// TIA Portal V16 export
// export: Created 2023-03-29T11:03:22.6082356Z, ExportSetting WithDefaults, DisplayName Totally Integrated Automation Portal, DisplayVersion V16 Update 6, DisplayName TIA Portal Version Control Interface, DisplayVersion V16 Update 2, DisplayName TIA Portal Openness, DisplayVersion V16 Update 6, DisplayName STEP 7 Professional, DisplayVersion V16 Update 6, DisplayName STEP 7 Safety, DisplayVersion V16, DisplayName WinCC Advanced, DisplayVersion V16 Update 6
FUNCTION "Sterowanie_Zbiornik" : Void   // FC26, LAD
TITLE = Napełnianie i opróżnianie
{ S7_Optimized_Access := 'TRUE' }
AUTHOR : rtecmer
VERSION : 0.1
// Funkcja steruje napędami napełniania i opróżniania w cyklu od zegara czasu jak i od pomiaru poziomu. Poziom jest sygnałem nadrzędnym. Jeśli napełnienie uzyskano przed czasem to napełnianie jest kończone z osiągnięciem poziomu max. Podczas oróżniania jeśli osiągnięto poziom min to opróżnianie zbiorniak jest zakończone.
// Granica końca minimum to 100cm ponad tę wartość nastąpi dopiero skasowanie sygnału poziom MIN
// Spadku poziomu poniżej 250cm pozwala na scasowanie sygnału poziom MAX
// stored: AutoNumber true, IsIECCheckEnabled false, SetENOAutomatically false, UDAEnableTagReadback false
   VAR_INPUT
      actLevel : Real;   // pozim w zbiorniku
      maxLevel : Real;   // poziom napełnienia
      minLevel : Real;   // poziom opróżnienia
      actTime : Real;   // czas aktualny
      actTime_FillingOn : Real;   // godzina start napełnianie
      actTime_FillingOff : Real;   // godzina stop napełnianie
      actTime_EmptyingOn : Real;   // godzina start przetłaczanie
      actTime_EmptyingOff : Real;   // godzina stop przetłaczanie
      isOpen_filling : Bool;   // potwierdzenie otwarcia napełniającej zasuwy
      isOpen_emptying : Bool;   // potwierdzenie otwarcia spustowej zasuwy
      isClose_filling : Bool;   // potwierdzenie zamknięcia napełniającej zasuwy
      isClose_emptying : Bool;   // potwierdzenie zamknięcia spustowej zasuwy
      isReady_filling : Bool;   // sygnał gotowości zasuwa napełnianie
      isReadyt_emptying : Bool;   // sygnał gotowości zasuwa spustowa
      activTank : Bool;   // zbiornik aktywny
      isAut_Valve_Filling : Bool;   // tryb pracy automat zasuwa napełnianie
      isAut_Valve_Empting : Bool;   // tryb pracy automat zasuwa spustowa
      is_min_Float : Bool;   // sygnał minimum z płyawaka
      is_max_Float : Bool;   // sygnał max z płyawaka
      isAlarmNinimum_barB5 : Bool;   // alarm niskie ciśnienie magistrala
      resetAlarmMinimum_barB5 : Bool;   // koniec alarm niskie ciśnienie magistral
      setTank_Work_daily : Bool;   // tryb pracy dobowy aktywny
      setTank_Work_selective : Bool;   // tryb pracy selektywny - jeden zbiornik aktywny
      setControl_alarm_B5 : Bool;   // sygnał uruchomienie awaryjnego otwarcie zbiornika na dosilanie
      set_HWork_tank : Bool;   // ustawia aktywny zbiornik do pracy w trybie selektywnym
   END_VAR
   VAR_OUTPUT
      setSVMO_Z_Wlot : Bool;   // bit otwierania w trybie automat
      setSVMC_Z_Wlot : Bool;   // bit zamykania w trybie automat
      setSVMO_Z_Spust : Bool;   // bit otwierania w trybie automat
      setSVMC_Z_Spust : Bool;   // bit zamykania w trybie automat
      infoFiling_to_HMI : Bool;   // bit informacji wejściu w tryb napełniania
   END_VAR
   VAR_IN_OUT
      isFilling : Bool;   // bit aktywacji napełninia
      isEptying : Bool;   // bit aktywacji przetłaczania
      memRisingLevel_min : Bool;   // pamięc zbocza osiągniecia poziomu minimum w zbiorniku
      memRisingLevel_max : Bool;   // pamięc zbocza osiągniecia poziomu max w zbiorniku
      isLevelMax : Bool;   // poziom max
      isLevelMin : Bool;   // poziom min
      blok_tank : Bool;   // bit blokowania zbiornika w sekwencji
   END_VAR
   VAR_TEMP
      correction_max : Real;   // współczynnik korekty dla zachowania histerezy przy wahaniu poziomu w zbiorniku
      correction_min : Real;   // współczynnik korekty dla zachowania histerezy przy wahaniu poziomu w zbiorniku
      filling_time : Real;   // wyliczony czas napełniania na dobę
      filing_time_X : Bool;   // bit logika gdy napełnianie przed 00:00
      filing_time_Y : Bool;   // bit logika gdy napełnianie po 00:01
      epting_time_X : Bool;   // bit logika gdy napełnianie po 00:01
   END_VAR
   VAR_TEMP   // added for the SCL form of the ladder/FBD networks
      _w1 : Bool;
      _w2 : Bool;
   END_VAR
BEGIN

REGION Network 1 (SCL): wyliczenie korekty dla stabilności sygału min i max
   #correction_max := (#maxLevel - 30);
   #correction_min := (#minLevel + 20);
END_REGION

REGION Network 2: znacznik poziom max
   // przechwycenie poziomu max
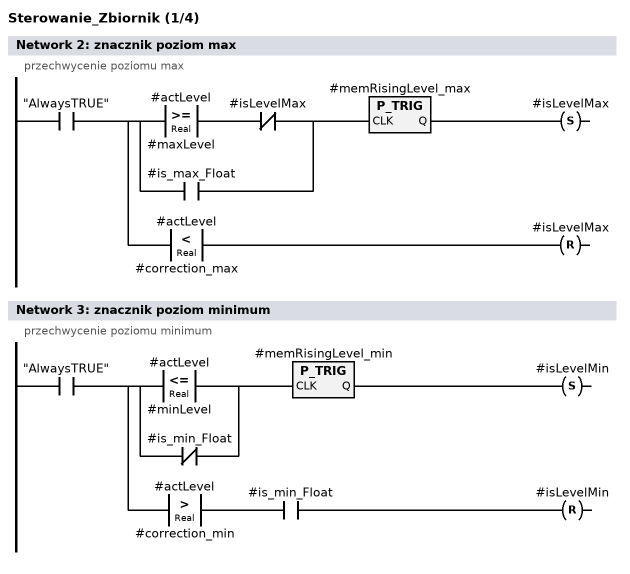
   RUNG wire#powerrail
      Contact( "AlwaysTRUE" )
      wire#w1
      { S7_Templates := "SrcType := Real" } GE_Contact(in1 := #actLevel, in2 := #maxLevel)
      I_Contact( #isLevelMax )
      wire#w2
      P_Trig( #memRisingLevel_max )
      S_Coil( #isLevelMax )
   END_RUNG
   RUNG wire#w1
      Contact( #is_max_Float )
   END_RUNG wire#w2
   RUNG wire#w1
      { S7_Templates := "SrcType := Real" } LT_Contact(in1 := #actLevel, in2 := #correction_max)
      R_Coil( #isLevelMax )
   END_RUNG
   // the same network as SCL:
   #_w1 := "AlwaysTRUE" AND (((#actLevel >= #maxLevel) AND NOT #isLevelMax) OR #is_max_Float);
   #_w2 := #_w1 AND NOT #memRisingLevel_max;   // rising edge
   #memRisingLevel_max := #_w1;
   IF #_w2 THEN #isLevelMax := TRUE; END_IF;
   IF "AlwaysTRUE" AND (#actLevel < #correction_max) THEN #isLevelMax := FALSE; END_IF;
END_REGION

REGION Network 3: znacznik poziom minimum
   // przechwycenie poziomu minimum
   RUNG wire#powerrail
      Contact( "AlwaysTRUE" )
      wire#w1
      { S7_Templates := "SrcType := Real" } LE_Contact(in1 := #actLevel, in2 := #minLevel)
      wire#w2
      P_Trig( #memRisingLevel_min )
      S_Coil( #isLevelMin )
   END_RUNG
   RUNG wire#w1
      I_Contact( #is_min_Float )
   END_RUNG wire#w2
   RUNG wire#w1
      { S7_Templates := "SrcType := Real" } GT_Contact(in1 := #actLevel, in2 := #correction_min)
      Contact( #is_min_Float )
      R_Coil( #isLevelMin )
   END_RUNG
   // the same network as SCL:
   #_w1 := "AlwaysTRUE" AND ((#actLevel <= #minLevel) OR NOT #is_min_Float);
   #_w2 := #_w1 AND NOT #memRisingLevel_min;   // rising edge
   #memRisingLevel_min := #_w1;
   IF #_w2 THEN #isLevelMin := TRUE; END_IF;
   IF "AlwaysTRUE" AND (#actLevel > #correction_min) AND #is_min_Float THEN #isLevelMin := FALSE; END_IF;
END_REGION

REGION Network 4 (SCL): wyliczony czas napełniania na dobę i ustawoanie bitu kontroli pracy w dobie
   // #filing_time_X  - bit ustawiany w przypadku gdy w przedziale pracy wystąpi przejście przez  godzinę 00:00
   IF #actTime_FillingOn > #actTime_FillingOff THEN
     // odejmnij od wiekszej mniejszą
     #filling_time := (#actTime_FillingOn - #actTime_FillingOff);
     IF #actTime >=  #actTime_FillingOn THEN
       // jeśli czas rozpoczęcia napełniania to ustaw bit
       #filing_time_X := TRUE;
       ;
     ELSE
       // w innym wypadku kasuj bit
       #filing_time_X := False;
       ;
     END_IF;

     #filing_time_Y := FALSE;
   ELSE
     #filling_time := (#actTime_FillingOff - #actTime_FillingOn);
     #filing_time_X := False;
     #filing_time_Y := TRUE;
     ;
   END_IF;
END_REGION

REGION Network 5: bit aktywacji napełninia
   // aktywacja, deaktywacja bitu rocedury napełniania
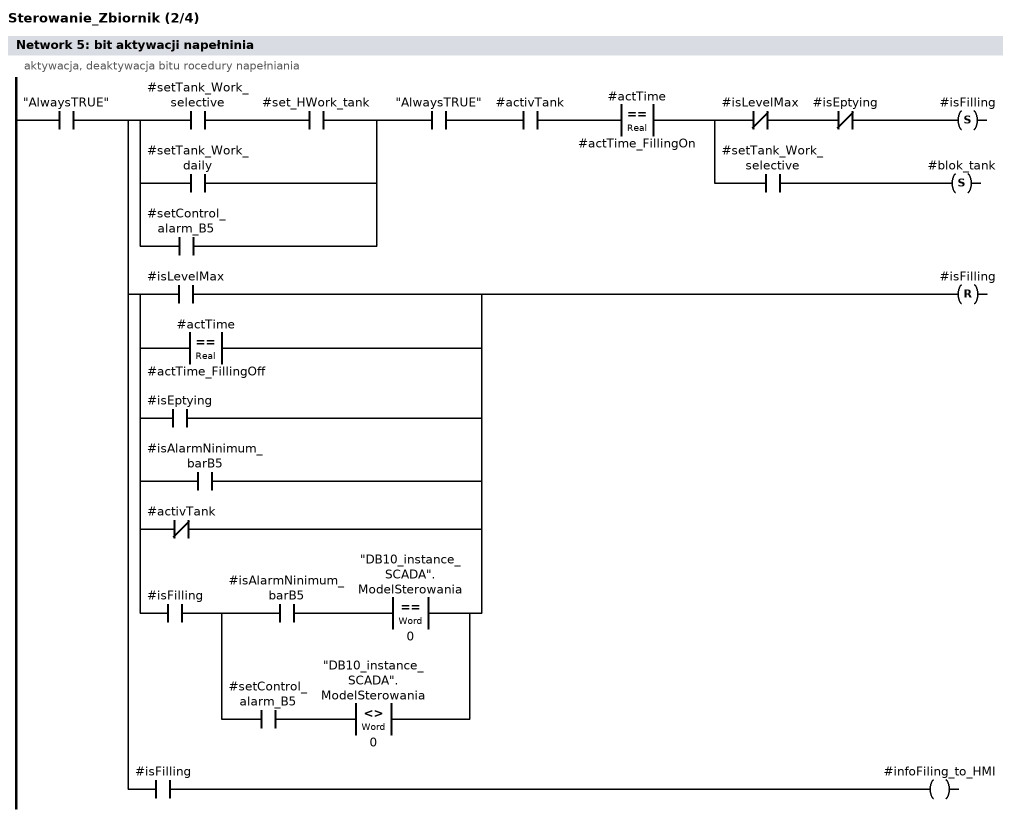
   RUNG wire#powerrail
      Contact( "AlwaysTRUE" )
      wire#w1
      Contact( #setTank_Work_selective )
      Contact( #set_HWork_tank )
      wire#w2
      Contact( "AlwaysTRUE" )
      Contact( #activTank )
      { S7_Templates := "SrcType := Real" } EQ_Contact(in1 := #actTime, in2 := #actTime_FillingOn)
      wire#w3
      I_Contact( #isLevelMax )
      I_Contact( #isEptying )
      S_Coil( #isFilling )
   END_RUNG
   RUNG wire#w1
      Contact( #setTank_Work_daily )
   END_RUNG wire#w2
   RUNG wire#w1
      Contact( #setControl_alarm_B5 )
   END_RUNG wire#w2
   RUNG wire#w3
      Contact( #setTank_Work_selective )
      S_Coil( #blok_tank )
   END_RUNG
   RUNG wire#w1
      Contact( #isLevelMax )
      wire#w4
      R_Coil( #isFilling )
   END_RUNG
   RUNG wire#w1
      { S7_Templates := "SrcType := Real" } EQ_Contact(in1 := #actTime, in2 := #actTime_FillingOff)
   END_RUNG wire#w4
   RUNG wire#w1
      Contact( #isEptying )
   END_RUNG wire#w4
   RUNG wire#w1
      Contact( #isAlarmNinimum_barB5 )
   END_RUNG wire#w4
   RUNG wire#w1
      I_Contact( #activTank )
   END_RUNG wire#w4
   RUNG wire#w1
      Contact( #isFilling )
      wire#w5
      Contact( #isAlarmNinimum_barB5 )
      { S7_Templates := "SrcType := Word" } EQ_Contact(in1 := "DB10_instance_SCADA".ModelSterowania, in2 := 0)
   END_RUNG wire#w4
   RUNG wire#w5
      Contact( #setControl_alarm_B5 )
      { S7_Templates := "SrcType := Word" } NE_Contact(in1 := "DB10_instance_SCADA".ModelSterowania, in2 := 0)
   END_RUNG wire#w4
   RUNG wire#w1
      Contact( #isFilling )
      Coil( #infoFiling_to_HMI )
   END_RUNG
   // the same network as SCL:
   #_w1 := "AlwaysTRUE" AND ((#setTank_Work_selective AND #set_HWork_tank) OR #setTank_Work_daily OR #setControl_alarm_B5) AND "AlwaysTRUE" AND #activTank AND (#actTime = #actTime_FillingOn);
   IF #_w1 AND NOT #isLevelMax AND NOT #isEptying THEN #isFilling := TRUE; END_IF;
   IF #_w1 AND #setTank_Work_selective THEN #blok_tank := TRUE; END_IF;
   IF "AlwaysTRUE" AND (#isLevelMax OR (#actTime = #actTime_FillingOff) OR #isEptying OR #isAlarmNinimum_barB5 OR NOT #activTank OR (#isFilling AND ((#isAlarmNinimum_barB5 AND ("DB10_instance_SCADA".ModelSterowania = 0)) OR (#setControl_alarm_B5 AND ("DB10_instance_SCADA".ModelSterowania <> 0))))) THEN
       #isFilling := FALSE;
   END_IF;
   #infoFiling_to_HMI := "AlwaysTRUE" AND #isFilling;
END_REGION

REGION Network 6 (SCL): ustawoanie bitu kontroli pracy w dobie
   // epting_time_X  - bit ustawiany w przypadku gdy w przedziale pracy wystąpi przejście przez  godzinę 00:00
   IF #actTime_EmptyingOn > #actTime_EmptyingOff THEN

     IF #actTime >=  #actTime_EmptyingOn THEN
       // jeśli czas rozpoczęcia napełniania to ustaw bit
       #epting_time_X := TRUE;
       ;
     ELSE
       // w innym wypadku kasuj bit
       #epting_time_X := False;
       ;
     END_IF;

   ELSE

     #epting_time_X := False;

     ;
   END_IF;
END_REGION

REGION Network 7: bit aktywacji przetłaczania
   // aktywacja/ deaktywacja bitu pracy pompowni (przetłaczanie)
   // musi zakonczyć się napełnianie, jeśli wyłaczysz z trybu automat to reset znacznika przetłaczanie
   // 
   // #epting_time_X - usunąłem na testy
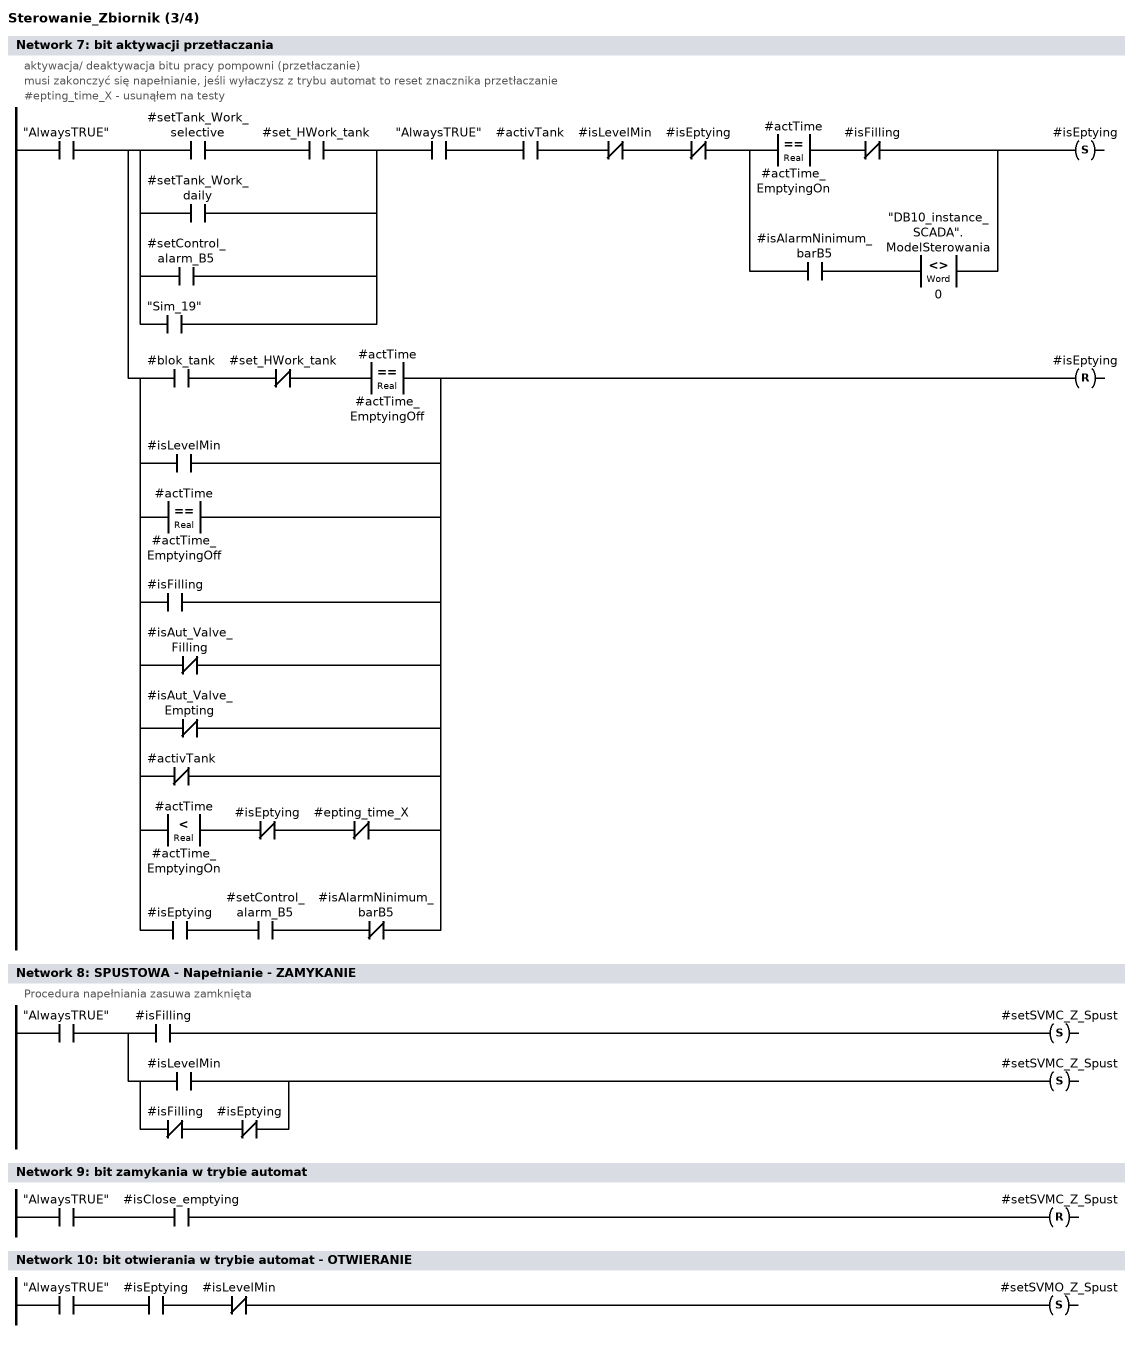
   RUNG wire#powerrail
      Contact( "AlwaysTRUE" )
      wire#w1
      Contact( #setTank_Work_selective )
      Contact( #set_HWork_tank )
      wire#w2
      Contact( "AlwaysTRUE" )
      Contact( #activTank )
      I_Contact( #isLevelMin )
      I_Contact( #isEptying )
      wire#w3
      { S7_Templates := "SrcType := Real" } EQ_Contact(in1 := #actTime, in2 := #actTime_EmptyingOn)
      I_Contact( #isFilling )
      wire#w4
      S_Coil( #isEptying )
   END_RUNG
   RUNG wire#w1
      Contact( #setTank_Work_daily )
   END_RUNG wire#w2
   RUNG wire#w1
      Contact( #setControl_alarm_B5 )
   END_RUNG wire#w2
   RUNG wire#w1
      Contact( "Sim_19" )
   END_RUNG wire#w2
   RUNG wire#w3
      Contact( #isAlarmNinimum_barB5 )
      { S7_Templates := "SrcType := Word" } NE_Contact(in1 := "DB10_instance_SCADA".ModelSterowania, in2 := 0)
   END_RUNG wire#w4
   RUNG wire#w1
      Contact( #blok_tank )
      I_Contact( #set_HWork_tank )
      { S7_Templates := "SrcType := Real" } EQ_Contact(in1 := #actTime, in2 := #actTime_EmptyingOff)
      wire#w5
      R_Coil( #isEptying )
   END_RUNG
   RUNG wire#w1
      Contact( #isLevelMin )
   END_RUNG wire#w5
   RUNG wire#w1
      { S7_Templates := "SrcType := Real" } EQ_Contact(in1 := #actTime, in2 := #actTime_EmptyingOff)
   END_RUNG wire#w5
   RUNG wire#w1
      Contact( #isFilling )
   END_RUNG wire#w5
   RUNG wire#w1
      I_Contact( #isAut_Valve_Filling )
   END_RUNG wire#w5
   RUNG wire#w1
      I_Contact( #isAut_Valve_Empting )
   END_RUNG wire#w5
   RUNG wire#w1
      I_Contact( #activTank )
   END_RUNG wire#w5
   RUNG wire#w1
      { S7_Templates := "SrcType := Real" } LT_Contact(in1 := #actTime, in2 := #actTime_EmptyingOn)
      I_Contact( #isEptying )
      I_Contact( #epting_time_X )
   END_RUNG wire#w5
   RUNG wire#w1
      Contact( #isEptying )
      Contact( #setControl_alarm_B5 )
      I_Contact( #isAlarmNinimum_barB5 )
   END_RUNG wire#w5
   // the same network as SCL:
   IF "AlwaysTRUE" AND ((#setTank_Work_selective AND #set_HWork_tank) OR #setTank_Work_daily OR #setControl_alarm_B5 OR "Sim_19") AND "AlwaysTRUE" AND #activTank AND NOT #isLevelMin AND NOT #isEptying AND (((#actTime = #actTime_EmptyingOn) AND NOT #isFilling) OR (#isAlarmNinimum_barB5 AND ("DB10_instance_SCADA".ModelSterowania <> 0))) THEN
       #isEptying := TRUE;
   END_IF;
   IF "AlwaysTRUE" AND ((#blok_tank AND NOT #set_HWork_tank AND (#actTime = #actTime_EmptyingOff)) OR #isLevelMin OR (#actTime = #actTime_EmptyingOff) OR #isFilling OR NOT #isAut_Valve_Filling OR NOT #isAut_Valve_Empting OR NOT #activTank OR ((#actTime < #actTime_EmptyingOn) AND NOT #isEptying AND NOT #epting_time_X) OR (#isEptying AND #setControl_alarm_B5 AND NOT #isAlarmNinimum_barB5)) THEN
       #isEptying := FALSE;
   END_IF;
END_REGION

REGION Network 8: SPUSTOWA - Napełnianie - ZAMYKANIE
   // Procedura napełniania zasuwa zamknięta
   RUNG wire#powerrail
      Contact( "AlwaysTRUE" )
      wire#w1
      Contact( #isFilling )
      S_Coil( #setSVMC_Z_Spust )
   END_RUNG
   RUNG wire#w1
      Contact( #isLevelMin )
      wire#w2
      S_Coil( #setSVMC_Z_Spust )
   END_RUNG
   RUNG wire#w1
      I_Contact( #isFilling )
      I_Contact( #isEptying )
   END_RUNG wire#w2
   // the same network as SCL:
   IF "AlwaysTRUE" AND #isFilling THEN #setSVMC_Z_Spust := TRUE; END_IF;
   IF "AlwaysTRUE" AND (#isLevelMin OR (NOT #isFilling AND NOT #isEptying)) THEN
       #setSVMC_Z_Spust := TRUE;
   END_IF;
END_REGION

REGION Network 9: bit zamykania w trybie automat
   RUNG wire#powerrail
      Contact( "AlwaysTRUE" )
      Contact( #isClose_emptying )
      R_Coil( #setSVMC_Z_Spust )
   END_RUNG
   // the same network as SCL:
   IF "AlwaysTRUE" AND #isClose_emptying THEN #setSVMC_Z_Spust := FALSE; END_IF;
END_REGION

REGION Network 10: bit otwierania w trybie automat - OTWIERANIE
   RUNG wire#powerrail
      Contact( "AlwaysTRUE" )
      Contact( #isEptying )
      I_Contact( #isLevelMin )
      S_Coil( #setSVMO_Z_Spust )
   END_RUNG
   // the same network as SCL:
   IF "AlwaysTRUE" AND #isEptying AND NOT #isLevelMin THEN #setSVMO_Z_Spust := TRUE; END_IF;
END_REGION

REGION Network 11: bit otwierania w trybie automat
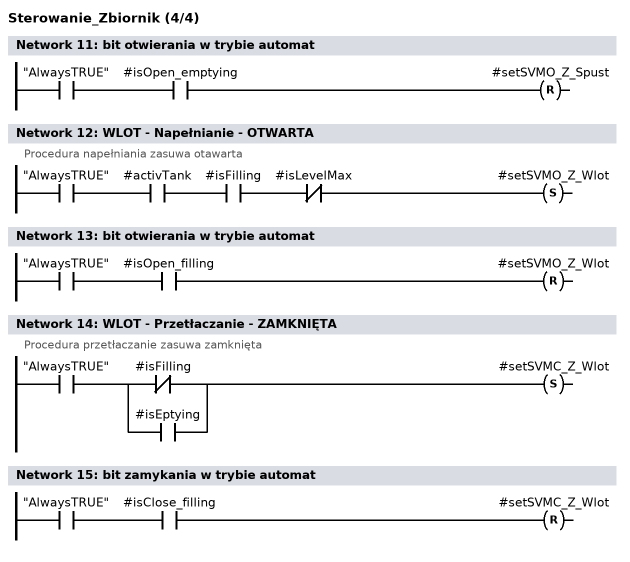
   RUNG wire#powerrail
      Contact( "AlwaysTRUE" )
      Contact( #isOpen_emptying )
      R_Coil( #setSVMO_Z_Spust )
   END_RUNG
   // the same network as SCL:
   IF "AlwaysTRUE" AND #isOpen_emptying THEN #setSVMO_Z_Spust := FALSE; END_IF;
END_REGION

REGION Network 12: WLOT - Napełnianie - OTWARTA
   // Procedura napełniania zasuwa otawarta
   RUNG wire#powerrail
      Contact( "AlwaysTRUE" )
      Contact( #activTank )
      Contact( #isFilling )
      I_Contact( #isLevelMax )
      S_Coil( #setSVMO_Z_Wlot )
   END_RUNG
   // the same network as SCL:
   IF "AlwaysTRUE" AND #activTank AND #isFilling AND NOT #isLevelMax THEN #setSVMO_Z_Wlot := TRUE; END_IF;
END_REGION

REGION Network 13: bit otwierania w trybie automat
   RUNG wire#powerrail
      Contact( "AlwaysTRUE" )
      Contact( #isOpen_filling )
      R_Coil( #setSVMO_Z_Wlot )
   END_RUNG
   // the same network as SCL:
   IF "AlwaysTRUE" AND #isOpen_filling THEN #setSVMO_Z_Wlot := FALSE; END_IF;
END_REGION

REGION Network 14: WLOT - Przetłaczanie - ZAMKNIĘTA
   // Procedura przetłaczanie zasuwa zamknięta
   RUNG wire#powerrail
      Contact( "AlwaysTRUE" )
      wire#w1
      I_Contact( #isFilling )
      wire#w2
      S_Coil( #setSVMC_Z_Wlot )
   END_RUNG
   RUNG wire#w1
      Contact( #isEptying )
   END_RUNG wire#w2
   // the same network as SCL:
   IF "AlwaysTRUE" AND (NOT #isFilling OR #isEptying) THEN #setSVMC_Z_Wlot := TRUE; END_IF;
END_REGION

REGION Network 15: bit zamykania w trybie automat
   RUNG wire#powerrail
      Contact( "AlwaysTRUE" )
      Contact( #isClose_filling )
      R_Coil( #setSVMC_Z_Wlot )
   END_RUNG
   // the same network as SCL:
   IF "AlwaysTRUE" AND #isClose_filling THEN #setSVMC_Z_Wlot := FALSE; END_IF;
END_REGION
END_FUNCTION
